Fanuc KAREL source: NC0083.KL

-- PROVISIONAL review KL for V770-1; original PC SHA256 57c40c3bd2860e3b8330a1e21479af8faf6cc49780adfe31aca4fbe11a503a19
-- Incomplete behavior may be omitted. Consult companion uncertainty JSON. Do not deploy.
PROGRAM NC0083
%NOLOCKGROUP
-- UNRESOLVED_LOCAL_POOL 1 cells at code offset 3; source declarations unknown
-- DIRECT_LOCAL_WORD_ACCESS alone does not prove INTEGER, REAL, or BOOLEAN
BEGIN
  -- UNRESOLVED_PC offsets 0-8; opcodes 2B,2C,7B
  -- UNRESOLVED_PC offsets 13-20; opcodes 9D,23
  -- UNRESOLVED_PC offsets 25-38; opcodes 21,9D,57,79
  -- UNRESOLVED_PC offsets 43-60; opcodes 21,40,41,42
  -- UNRESOLVED_PC offsets 65-95; opcodes 21,9D,52,23,7A,40,41,42
  -- UNRESOLVED_PC offsets 100-124; opcodes 21,2E,52,23,7A,43
  -- UNRESOLVED_PC offsets 129-147; opcodes 21,2E,52,23
  -- UNRESOLVED_PC offsets 157-162; opcodes 7A
  -- UNRESOLVED_PC offsets 167-185; opcodes 21,2E,52,23
  -- UNRESOLVED_PC offsets 195-199; opcodes 7F
  -- UNRESOLVED_PC offsets 204-208; opcodes 27,AA
  -- UNRESOLVED_PC offsets 213-217; opcodes 7F
END NC0083
